FUNCTION_BLOCK PNP_CTL_LD (* Pick and Place AUTO Control with LD Algorithm *)
  (* Standard: IEC 61499; ApplicationDomain: Discrete Assembly; Function: Pick&Place *)
  (* Version 0.2, 2006-09-16, JHC, Holobloc Inc, Converted to SimpleFB. *)
  (* Version 0.1, 2006-07-07, JHC, Holobloc Inc, Added LOADED sensor + associated logic. *)
  (* Version 0.0, 2006-06-26, JHC, Holobloc Inc, Updated sensor/actuator names and state machine *)
  (* Compiler header: package fb.rt.mach; *)
  (* Compiler classdef: SimpleFB *)
  (* Compiler Java Sun JDK 1.5.0 *)
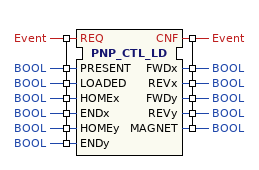
  EVENT_INPUT
    REQ WITH HOMEx, ENDx, HOMEy, ENDy, PRESENT, LOADED; (* Execute control if AUTO mode is ON *)
  END_EVENT
  EVENT_OUTPUT
    CNF WITH FWDx, FWDy, REVy, REVx, MAGNET; (* AUTO mode control executed *)
  END_EVENT
  VAR_INPUT
    PRESENT : BOOL; (* Workpiece Sensor at end of Conveyor *)
    LOADED : BOOL; (* Workpiece Sensor on XY transport *)
    HOMEx : BOOL; (* x-axis at HOME position *)
    ENDx : BOOL; (* x-axis at END position *)
    HOMEy : BOOL; (* y-axis at HOME position *)
    ENDy : BOOL; (* y-axis at END position *)
  END_VAR
  VAR_OUTPUT
    FWDx : BOOL; (* Drive x-axis Motor Forward (toward ENDx) *)
    REVx : BOOL; (* Drive x-axis Motor 1 in Reverse (toward HOMEx) *)
    FWDy : BOOL; (* Drive y-axis Motor Forward (toward ENDy) *)
    REVy : BOOL; (* Drive y-axis Motor 2 in Reverse (toward HOMEy) *)
    MAGNET : BOOL; (* Electromagnet ON (grasp workpiece) *)
  END_VAR
  ALGORITHM REQ IN LD: (* AUTO control algorithm *)
    MAGNET := PRESENT LOADED ! & HOMEx & HOMEy  & LOADED ENDx ! ENDy ! | & |;
    FWDx := LOADED ENDx ! &;
    FWDy := LOADED ENDx & ENDy ! &;
    REVx := LOADED ! HOMEx ! &;
    REVy := LOADED ! HOMEy ! &;
  END_ALGORITHM
END_FUNCTION_BLOCK
